(* PLC project PLCopen TC4 OPC UA, University of Seoul OPC UA 0.0 *)
(* stored: creationDateTime 2015-10-01T00:00:00, modificationDateTime 2015-10-01T00:00:00 *)

TYPE UASecurityMsgMode : (UASMM_BestAvailable, UASMM_None, UASMM_Sign, UASMM_SignEncrypt);
END_TYPE

TYPE UASecurityPolicy : (UASP_BestAvailable, UASP_None, UASP_Basic128Rsa15, UASP_Basic256, UASP_Basic256Sha256);
END_TYPE

TYPE UATransportProfile : (UATP_UATcp, UATP_WSHttpBinary, UATP_WSHttpXmlOrBinary, UATP_WSHttpXml);
END_TYPE

TYPE UAUserIdentityTokenType : (UAUITT_Anonymous, UAUITT_Username, UAUITT_x509, UAUITT_IssuedToken);
END_TYPE

TYPE UAIdentifierType : (UAIT_Numeric, UAIT_String, UAIT_GUID, UAIT_Opaque);
END_TYPE

TYPE UADeadbandType : (UADT_None, UADT_Absolute, UADT_Percent) := UADT_None;
END_TYPE

TYPE UAAttributeID : (UAAI_NodeID, UAAI_NodeClass, UAAI_BrowseName, UAAI_DisplayName, UAAI_Description, UAAI_WriteMask, UAAI_UserWriteMask, UAAI_IsAbstract, UAAI_Symmetric, UAAI_InverseName, UAAI_ContainsNoLoops, UAAI_EventNotifier, UAAI_Value, UAAI_DataType, UAAI_ValueRank, UAAI_ArrayDimensions, UAAI_AccessLevel, UAAI_UserAccessLevel, UAAI_MinimumSamplingInterval, UAAI_Historizing, UAAI_Executable, UAAI_UserExecutable) := UAAI_NodeID;
END_TYPE

TYPE UAConnectionStatus : (UACS_Connected, UACS_ConnectionError, UACS_Shutdown);
END_TYPE

TYPE UAServerState : (UASS_Running, UASS_Failed, UASS_NoConfiguration, UASS_Suspended, UASS_Shutdown, UASS_Test, UASS_CommunicationFault, UASS_Unknown);
END_TYPE

TYPE UANodeClassMask : (UANCM_None, UANCM_Object, UANCM_Variable, UANCM_Method, UANCM_ObjectType, UANCM_VariableType, UANCM_ReferenceType, UANCM_DataType, UANCM_View, UANCM_All);
END_TYPE

TYPE _UA_VariantType : (PlcOpen_VariantType_Boolaen, PlcOpen_VariantType_Byte, PlcOpen_VariantType_CharA, PlcOpen_VariantType_Int16, PlcOpen_VariantType_Int32, PlcOpen_VariantType_UInt16, PlcOpen_VariantType_UInt32, PlcOpen_VariantType_Double, PlcOpen_VariantType_Float, PlcOpen_VariantType_StringA, PlcOpen_VariantType_DateTime, PlcOpen_VariantType_QualifiedName);
END_TYPE

TYPE UAUserIdentityToken : STRUCT
  UserIdentityTokenType : UAUserIdentityTokenType;
  TokenParam1 : STRING;
  TokenParam2 : STRING;
END_STRUCT;
END_TYPE

TYPE UASessionConnectInfo : STRUCT
  SessionName : STRING;
  ApplicationName : STRING;
  SecurityMsgMode : UASecurityMsgMode;
  SecurityPolicy : UASecurityPolicy;
  CertificateStore : STRING;
  ClientCertificateName : STRING;
  ServerUri : STRING;
  CheckServerCertificate : BOOL;
  TransportProfile : UATransportProfile;
  UserIdentityToken : UAUserIdentityToken;
  VendorSpecificParameter : STRING;
  SessionTimeout : STRING;
  MonitorConnection : STRING;
  LocaleIDs : STRING;
END_STRUCT;
END_TYPE

TYPE UANODEID : STRUCT
  NamespaceIndex : UINT;
  Identifier : STRING;
  IdentifierType : UAIdentifierType;
END_STRUCT;
END_TYPE

TYPE UAQualifiedName : STRUCT
  NamespaceIndex : UINT;
  Name : STRING;
END_STRUCT;
END_TYPE

TYPE UAMONITORINGPARAMETER : STRUCT
  SamplingInterval : STRING;
  QueueSize : UINT;
  DiscardOldest : BOOL;
  DeadbandType : UADeadbandType;
  Deadband : REAL;
END_STRUCT;
END_TYPE

TYPE UALocalizedText : STRUCT
  Locale : _UALocaleType;
  Text : STRING;
END_STRUCT;
END_TYPE

TYPE UANodeInformation : STRUCT
  AccessLevel : BYTE;
  ArrayDimension : _UA_UDINT_ArrayType;
  BrowseName : UAQualifiedName;
  ContainsNoLoops : BOOL;
  DataType : UANODEID;
  Description : UALocalizedText;
  DisplayName : UALocalizedText;
  EventNotifier : BYTE;
  Executable : BOOL;
  Historizing : BOOL;
  InverseName : STRING;
  IsAbstract : BOOL;
  MinimumSamplingInterval : STRING;
  NodeClass : UANodeClassMask;
  Symmetric : BOOL;
  UserAccessLevel : BYTE;
  UserExecutable : BOOL;
  UserWriteMask : UDINT;
  ValueRank : DINT;
  WriteMask : UDINT;
END_STRUCT;
END_TYPE

TYPE UAINDEXRANGE : STRUCT
  StartIndex : UINT;
  EndIndex : UINT;
END_STRUCT;
END_TYPE

TYPE UANODEADDITIONALINFO : STRUCT
  AttributeID : UAAttributeID;
  IndexRangeCount : UINT;
  IndexRange : ARRAY[1..20] OF UAINDEXRANGE;
END_STRUCT;
END_TYPE

TYPE _UA_BOOL_ArrayType : STRUCT
  Elements : ARRAY[1..20] OF BOOL;
END_STRUCT;
END_TYPE

TYPE _UA_UINT_ArrayType : STRUCT
  Elements : ARRAY[1..20] OF UINT;
END_STRUCT;
END_TYPE

TYPE _UA_UDINT_ArrayType : STRUCT
  Elements : ARRAY[1..20] OF UDINT;
END_STRUCT;
END_TYPE

TYPE _UA_DT_ArrayType : STRUCT
  Elements : ARRAY[1..20] OF STRING;
END_STRUCT;
END_TYPE

TYPE _UA_STRING_ArrayType : STRUCT
  Elements : ARRAY[1..20] OF STRING;
END_STRUCT;
END_TYPE

TYPE _UA_DWORD_ArrayType : STRUCT
  Elements : ARRAY[1..20] OF DWORD;
END_STRUCT;
END_TYPE

TYPE _UA_UANODEID_ArrayType : STRUCT
  Elements : ARRAY[1..20] OF UANODEID;
END_STRUCT;
END_TYPE

TYPE _UA_MONITORINGPARAMETER_ArrayType : STRUCT
  Elements : ARRAY[1..20] OF UAMONITORINGPARAMETER;
END_STRUCT;
END_TYPE

TYPE _UA_NODEADDITIONALINFO_ArrayType : STRUCT
  Elements : ARRAY[1..20] OF UANODEADDITIONALINFO;
END_STRUCT;
END_TYPE

TYPE _UA_METHODARGUMENT_ArrayType : STRUCT
  Elements : ARRAY[1..20] OF _UA_METHODARGUMENT;
END_STRUCT;
END_TYPE

TYPE _UALocaleType : STRUCT
  Locale : ARRAY[1..5] OF STRING;
END_STRUCT;
END_TYPE

TYPE _UA_METHODARGUMENT : STRUCT
  VariantType : _UA_VariantType;
  Value : STRING;
END_STRUCT;
END_TYPE

TYPE _UA_MethodParameter : STRUCT
  NoOfArgument : UINT;
  Arguments : _UA_METHODARGUMENT_ArrayType;
END_STRUCT;
END_TYPE

FUNCTION_BLOCK UA_Connect
  VAR_INPUT
    Execute : BOOL := FALSE;
    ServerEndpointUrl : STRING;
    SessionConnectInfo : UASessionConnectInfo;
    Timeout : TIME;
  END_VAR
  VAR_OUTPUT
    ConnectionHdl : DWORD;
    Done : BOOL := FALSE;
    Busy : BOOL := FALSE;
    Error : BOOL := FALSE;
    ErrorID : DWORD;
  END_VAR
  VAR
    State : DWORD;
    Trigm1 : BOOL := FALSE;
    Trigged : BOOL := FALSE;
    Pre_ServerEndpointUrl : STRING;
    Pre_ServerEndpointUrl0 : STRING;
    Pre_SessionConnectInfo : UASessionConnectInfo;
    Pre_SessionConnectInfo0 : UASessionConnectInfo;
    Pre_Timeout : TIME;
    Pre_Timeout0 : TIME;
    Pre_ConnectionHdl : DWORD;
    Pre_ErrorID : DWORD;
  END_VAR

{{
  #ifdef _ENABLE_OPC_UA_CLIENT
  extern void __UA_ConnectFB(UA_CONNECT*);
  __UA_ConnectFB(data__);
  #endif
}}
          
END_FUNCTION_BLOCK

FUNCTION_BLOCK UA_Disconnect
  VAR_INPUT
    Execute : BOOL;
    ConnectionHdl : DWORD;
    Timeout : TIME;
  END_VAR
  VAR_OUTPUT
    Done : BOOL;
    Busy : BOOL;
    Error : BOOL;
    ErrorID : DWORD;
  END_VAR
  VAR
    State : DWORD;
    Trigm1 : BOOL;
    Trigged : BOOL;
    Pre_ConnectionHdl : DWORD;
    Pre_ConnectionHdl0 : DWORD;
    Pre_Timeout : TIME;
    Pre_Timeout0 : TIME;
    Pre_ErrorID : DWORD;
  END_VAR

{{
  #ifdef _ENABLE_OPC_UA_CLIENT
  extern void __UA_DisconnectFB(UA_DISCONNECT*);
  __UA_DisconnectFB(data__);
  #endif
}}
          
END_FUNCTION_BLOCK

FUNCTION_BLOCK UA_NamespaceGetIndexList
  VAR_INPUT
    Execute : BOOL;
    ConnectionHdl : DWORD;
    NamespaceUrisCount : UINT;
    NamespaceUris : _UA_STRING_ArrayType;
    Timeout : TIME;
  END_VAR
  VAR_OUTPUT
    NamespaceIndexes : _UA_UINT_ArrayType;
    Done : BOOL;
    Busy : BOOL;
    Error : BOOL;
    ErrorID : DWORD;
    ErrorIDs : ARRAY[1..50] OF DWORD;
  END_VAR
  VAR
    State : DWORD;
    Trigm1 : BOOL;
    Trigged : BOOL;
    Pre_ConnectionHdl : DWORD;
    Pre_ConnectionHdl0 : DWORD;
    Pre_NamespaceUrisCount : UINT;
    Pre_NamespaceUrisCount0 : UINT;
    Pre_NamespaceUris : _UA_STRING_ArrayType;
    Pre_NamespaceUris0 : _UA_STRING_ArrayType;
    Pre_NamespaceIndexes : _UA_UINT_ArrayType;
    Pre_Timeout : TIME;
    Pre_Timeout0 : TIME;
    Pre_ErrorID : DWORD;
  END_VAR

{{
  #ifdef _ENABLE_OPC_UA_CLIENT
  extern void __UA_NamespaceGetIndexListFB(UA_NAMESPACEGETINDEXLIST*);
  __UA_NamespaceGetIndexListFB(data__);
  #endif
}}
          
END_FUNCTION_BLOCK

FUNCTION_BLOCK UA_NodeGetHandleList
  VAR_INPUT
    Execute : BOOL;
    ConnectionHdl : DWORD;
    NodeIDCount : UINT;
    NodeIDs : _UA_UANODEID_ArrayType;
    Timeout : TIME;
  END_VAR
  VAR_OUTPUT
    NodeHdls : _UA_DWORD_ArrayType;
    Done : BOOL;
    Busy : BOOL;
    Error : BOOL;
    ErrorID : DWORD;
    NodeErrorIDs : ARRAY[1..20] OF DWORD;
  END_VAR
  VAR
    State : DWORD;
    Trigm1 : BOOL;
    Trigged : BOOL;
    Pre_ConnectionHdl : DWORD;
    Pre_ConnectionHdl0 : DWORD;
    Pre_NodeIDCount : UINT;
    Pre_NodeIDCount0 : UINT;
    Pre_NodeIDs : _UA_UANODEID_ArrayType;
    Pre_NodeIDs0 : _UA_UANODEID_ArrayType;
    Pre_Timeout : TIME;
    Pre_Timeout0 : TIME;
    Pre_NodeHdls : _UA_DWORD_ArrayType;
    Pre_ErrorID : DWORD;
    Pre_NodeErrorIDs : ARRAY[1..20] OF DWORD;
  END_VAR

{{
  #ifdef _ENABLE_OPC_UA_CLIENT
  extern void __UA_NodeGetHandleListFB(UA_NODEGETHANDLELIST*);
  __UA_NodeGetHandleListFB(data__);
  #endif
}}
          
END_FUNCTION_BLOCK

FUNCTION_BLOCK UA_NodeReleaseHandleList
  VAR_INPUT
    Execute : BOOL;
    ConnectionHdl : DWORD;
    NodeHdlCount : UINT;
    NodeHdls : _UA_DWORD_ArrayType;
    Timeout : TIME;
  END_VAR
  VAR_OUTPUT
    Done : BOOL;
    Busy : BOOL;
    Error : BOOL;
    ErrorID : DWORD;
    NodeErrorIDs : ARRAY[1..20] OF DWORD;
  END_VAR
  VAR
    State : DWORD;
    Trigm1 : BOOL;
    Trigged : BOOL;
    Pre_ConnectionHdl : DWORD;
    Pre_ConnectionHdl0 : DWORD;
    Pre_NodeHdlCount : UINT;
    Pre_NodeHdlCount0 : UINT;
    Pre_NodeHdls : _UA_DWORD_ArrayType;
    Pre_NodeHdls0 : _UA_DWORD_ArrayType;
    Pre_Timeout : TIME;
    Pre_Timeout0 : TIME;
    Pre_ErrorID : DWORD;
    Pre_NodeErrorIDs : ARRAY[1..20] OF DWORD;
  END_VAR

{{
  #ifdef _ENABLE_OPC_UA_CLIENT
  extern void __UA_NodeReleaseHandleListFB(UA_NODERELEASEHANDLELIST*);
  __UA_NodeReleaseHandleListFB(data__);
  #endif
}}
          
END_FUNCTION_BLOCK

FUNCTION_BLOCK UA_NodeGetInformation
  VAR_INPUT
    Execute : BOOL;
    ConnectionHdl : DWORD;
    NodeID : UANODEID;
    Timeout : TIME;
  END_VAR
  VAR_OUTPUT
    NodeInfo : UANodeInformation;
    Done : BOOL;
    Busy : BOOL;
    Error : BOOL;
    NodeGetInfoErrorIDs : ARRAY[0..21] OF DWORD;
  END_VAR
  VAR
    State : BOOL;
    Trigm1 : BOOL;
    Trigged : BOOL;
    Pre_ConnectionHdl : DWORD;
    Pre_ConnectionHdl0 : DWORD;
    Pre_NodeID : UANODEID;
    Pre_NodeID0 : UANODEID;
    Pre_Timeout : TIME;
    Pre_Timeout0 : TIME;
    Pre_NodeInfo : UANodeInformation;
    Pre_NodeGetInfoErrorIDs : ARRAY[0..21] OF DWORD;
    ErrorID : DWORD;
  END_VAR

{{
  #ifdef _ENABLE_OPC_UA_CLIENT
  extern void __UA_NodeGetInformationFB(UA_NODEGETINFORMATION*);
  __UA_NodeGetInformationFB(data__);
  #endif
}}
          
END_FUNCTION_BLOCK

FUNCTION_BLOCK UA_SubscriptionCreate
  VAR_INPUT
    Execute : BOOL;
    ConnectionHdl : DWORD;
    PublishingEnable : BOOL;
    Priority : BYTE;
    Timeout : TIME;
  END_VAR
  VAR_OUTPUT
    SubscriptionHdl : DWORD;
    Done : BOOL;
    Busy : BOOL;
    Error : BOOL;
    ErrorID : DWORD;
  END_VAR
  VAR_IN_OUT
    PublishingInterval : TIME;
  END_VAR
  VAR
    State : DWORD;
    Trigm1 : BOOL;
    Trigged : BOOL;
    Pre_ConnectionHdl : DWORD;
    Pre_ConnectionHdl0 : DWORD;
    Pre_PublishingEnable : BOOL;
    Pre_PublishingEnable0 : BOOL;
    Pre_Priority : BYTE;
    Pre_Priority0 : BYTE;
    Pre_Timeout : TIME;
    Pre_Timeout0 : TIME;
    Pre_PublishingInterval : TIME;
    Pre_PublishingInterval0 : TIME;
    Pre_PublishingInterval1 : TIME;
    Pre_SubscriptionHdl : DWORD;
    Pre_SubscriptionHdl0 : DWORD;
    Pre_ErrorID : DWORD;
    Pre_ErrorID0 : DWORD;
  END_VAR

{{
  #ifdef _ENABLE_OPC_UA_CLIENT
  extern void __UA_SubscriptionCreateFB(UA_SUBSCRIPTIONCREATE*);
  __UA_SubscriptionCreateFB(data__);
  #endif
}}
          
END_FUNCTION_BLOCK

FUNCTION_BLOCK UA_SubscriptionDelete
  VAR_INPUT
    Execute : BOOL;
    SubscriptionHdl : DWORD;
    Timeout : TIME;
  END_VAR
  VAR_OUTPUT
    Done : BOOL;
    Busy : BOOL;
    Error : BOOL;
    ErrorID : DWORD;
  END_VAR
  VAR
    State : DWORD;
    Trigm1 : BOOL;
    Trigged : BOOL;
    Pre_SubscriptionHdl : DWORD;
    Pre_SubscriptionHdl0 : DWORD;
    Pre_Timeout : TIME;
    Pre_Timeout0 : TIME;
    Pre_ErrorID : DWORD;
  END_VAR

{{
  #ifdef _ENABLE_OPC_UA_CLIENT
  extern void __UA_SubscriptionDeleteFB(UA_SUBSCRIPTIONDELETE*);
  __UA_SubscriptionDeleteFB(data__);
  #endif

}}
          
END_FUNCTION_BLOCK

FUNCTION_BLOCK UA_SubscriptionProcessed
  VAR_INPUT
    Execute : BOOL;
    SubscriptionHdl : DWORD;
  END_VAR
  VAR
    Pre_SubscriptionHdl : DWORD;
    Pre_SubscriptionHdl0 : DWORD;
  END_VAR
  VAR_INPUT
    Timeout : TIME;
  END_VAR
  VAR
    Pre_Timeout : TIME;
    Pre_Timeout0 : TIME;
  END_VAR
  VAR_OUTPUT
    Published : BOOL;
  END_VAR
  VAR
    Pre_Published : BOOL;
  END_VAR
  VAR_OUTPUT
    Done : BOOL;
    Busy : BOOL;
    Error : BOOL;
    ErrorID : DWORD;
  END_VAR
  VAR
    Pre_ErrorID : DWORD;
    State : DWORD;
    Trigged : BOOL;
    Trigm1 : BOOL;
  END_VAR

{{
  #ifdef _ENABLE_OPC_UA_CLIENT
  extern void __UA_SubscriptionProcessedFB(UA_SUBSCRIPTIONPROCESSED*);
  __UA_SubscriptionProcessedFB(data__);
  #endif
}}
          
END_FUNCTION_BLOCK

FUNCTION_BLOCK UA_MonitoredItemAddList
  VAR_INPUT
    Execute : BOOL;
    SubscriptionHdl : DWORD;
  END_VAR
  VAR
    Pre_SubscriptionHdl : DWORD;
    Pre_SubscriptionHdl0 : DWORD;
  END_VAR
  VAR_INPUT
    NodeHdlCount : UINT;
  END_VAR
  VAR
    Pre_NodeHdlCount : UINT;
    Pre_NodeHdlCount0 : UINT;
  END_VAR
  VAR_INPUT
    NodeHdls : _UA_DWORD_ArrayType;
  END_VAR
  VAR
    Pre_NodeHdls : _UA_DWORD_ArrayType;
    Pre_NodeHdls0 : _UA_DWORD_ArrayType;
  END_VAR
  VAR_INPUT
    NodeAddInfos : _UA_NodeAdditionalInfo_ArrayType;
  END_VAR
  VAR
    Pre_NodeAddInfos : _UA_NodeAdditionalInfo_ArrayType;
    Pre_NodeAddInfos0 : _UA_NodeAdditionalInfo_ArrayType;
  END_VAR
  VAR_INPUT
    Timeout : TIME;
  END_VAR
  VAR
    Pre_Timeout : TIME;
    Pre_Timeout0 : TIME;
  END_VAR
  VAR_OUTPUT
    Done : BOOL;
    Busy : BOOL;
    Error : BOOL;
    ErrorID : DWORD;
  END_VAR
  VAR
    Pre_ErrorID : DWORD;
  END_VAR
  VAR_OUTPUT
    NodeErrorIDs : _UA_DWORD_ArrayType;
  END_VAR
  VAR
    Pre_NodeErrorIDs : _UA_DWORD_ArrayType;
  END_VAR
  VAR_OUTPUT
    MonitoredItemHdls : _UA_DWORD_ArrayType;
  END_VAR
  VAR
    Pre_MonitoredItemHdls : _UA_DWORD_ArrayType;
  END_VAR
  VAR_IN_OUT
    Variables : UINT;
  END_VAR
  VAR
    Pre_Variables : UINT;
    Pre_Variables0 : UINT;
    Pre_Variables1 : UINT;
  END_VAR
  VAR_IN_OUT
    MonitoringSettings : _UA_MONITORINGPARAMETER_ArrayType;
  END_VAR
  VAR
    Pre_MonitoringSettings : _UA_MONITORINGPARAMETER_ArrayType;
    Pre_MonitoringSettings0 : _UA_MONITORINGPARAMETER_ArrayType;
    Pre_MonitoringSettings1 : _UA_MONITORINGPARAMETER_ArrayType;
  END_VAR
  VAR_IN_OUT
    ValuesChanged : UINT;
  END_VAR
  VAR
    Pre_ValuesChanged : UINT;
    Pre_ValuesChanged0 : UINT;
    Pre_ValuesChanged1 : UINT;
  END_VAR
  VAR_IN_OUT
    RemainingValueCount : _UA_UINT_ArrayType;
  END_VAR
  VAR
    Pre_RemainingValueCount : _UA_UINT_ArrayType;
    Pre_RemainingValueCount0 : _UA_UINT_ArrayType;
    Pre_RemainingValueCount1 : _UA_UINT_ArrayType;
  END_VAR
  VAR_IN_OUT
    TimeStamps : _UA_DT_ArrayType;
  END_VAR
  VAR
    Pre_TimeStamps : _UA_DT_ArrayType;
    Pre_TimeStamps0 : _UA_DT_ArrayType;
    Pre_TimeStamps1 : _UA_DT_ArrayType;
  END_VAR
  VAR_IN_OUT
    NodeQualityIDs : _UA_DWORD_ArrayType;
  END_VAR
  VAR
    Pre_NodeQualityIDs : _UA_DWORD_ArrayType;
    Pre_NodeQualityIDs0 : _UA_DWORD_ArrayType;
    Pre_NodeQualityIDs1 : _UA_DWORD_ArrayType;
    State : DWORD;
    Trigm1 : BOOL;
    Trigged : BOOL;
  END_VAR

{{
  #ifdef _ENABLE_OPC_UA_CLIENT
  extern void __UA_MonitoredItemAddListFB(UA_MONITOREDITEMADDLIST*);
  __UA_MonitoredItemAddListFB(data__);
  #endif
}}
          
END_FUNCTION_BLOCK

FUNCTION_BLOCK UA_MonitoredItemRemoveList
  VAR_INPUT
    Execute : BOOL;
    SubscriptionHdl : DWORD;
  END_VAR
  VAR
    Pre_SubscriptionHdl : DWORD;
    Pre_SubscriptionHdl0 : DWORD;
  END_VAR
  VAR_INPUT
    MonitoredItemHdlCount : UINT;
  END_VAR
  VAR
    Pre_MonitoredItemHdlCount : UINT;
    Pre_MonitoredItemHdlCount0 : UINT;
  END_VAR
  VAR_INPUT
    MonitoredItemHdls : _UA_DWORD_ArrayType;
  END_VAR
  VAR
    Pre_MonitoredItemHdls : _UA_DWORD_ArrayType;
    Pre_MonitoredItemHdls0 : _UA_DWORD_ArrayType;
  END_VAR
  VAR_INPUT
    Timeout : TIME;
  END_VAR
  VAR
    Pre_Timeout : TIME;
    Pre_Timeout0 : TIME;
  END_VAR
  VAR_OUTPUT
    Done : BOOL;
    Busy : BOOL;
    Error : BOOL;
    ErrorID : DWORD;
  END_VAR
  VAR
    Pre_ErrorID : DWORD;
  END_VAR
  VAR_OUTPUT
    NodeErrorIDs : _UA_DWORD_ArrayType;
  END_VAR
  VAR
    Pre_NodeErrorIDs : _UA_DWORD_ArrayType;
    State : DWORD;
    Trigm1 : BOOL;
    Trigged : BOOL;
  END_VAR

{{
  #ifdef _ENABLE_OPC_UA_CLIENT
  extern void __UA_MonitoredItemRemoveListFB(UA_MONITOREDITEMREMOVELIST*);
  __UA_MonitoredItemRemoveListFB(data__);
  #endif
}}
          
END_FUNCTION_BLOCK

FUNCTION_BLOCK UA_MonitoredItemOperateList
  VAR_INPUT
    Enable : BOOL;
    SubscriptionHdl : DWORD;
  END_VAR
  VAR
    Pre_SubscriptionHdl : DWORD;
    Pre_SubscriptionHdl0 : DWORD;
  END_VAR
  VAR_INPUT
    MonitoredItemHdlCount : UINT;
  END_VAR
  VAR
    Pre_MonitoredItemHdlCount : UINT;
    Pre_MonitoredItemHdlCount0 : UINT;
  END_VAR
  VAR_INPUT
    MonitoredItemHdls : _UA_DWORD_ArrayType;
  END_VAR
  VAR
    Pre_MonitoredItemHdls : _UA_DWORD_ArrayType;
    Pre_MonitoredItemHdls0 : _UA_DWORD_ArrayType;
  END_VAR
  VAR_OUTPUT
    Published : BOOL;
  END_VAR
  VAR
    Pre_Published : BOOL;
  END_VAR
  VAR_OUTPUT
    Done : BOOL;
    Busy : BOOL;
    Error : BOOL;
    ErrorID : DWORD;
  END_VAR
  VAR
    Pre_ErrorID : DWORD;
    State : DWORD;
    Trigm1 : BOOL;
    Trigged : BOOL;
  END_VAR

{{
  #ifdef _ENABLE_OPC_UA_CLIENT
  extern void __UA_MonitoredItemOperateListFB(UA_MONITOREDITEMOPERATELIST*);
  __UA_MonitoredItemOperateListFB(data__);
  #endif
}}
          
END_FUNCTION_BLOCK

FUNCTION_BLOCK UA_ReadList
  VAR_INPUT
    Execute : BOOL;
    ConnectionHdl : DWORD;
    NodeHdlCount : UINT;
    NodeHdls : _UA_DWORD_ArrayType;
    NodeAddInfos : ARRAY[1..20] OF UANODEADDITIONALINFO;
    Timeout : TIME;
  END_VAR
  VAR_OUTPUT
    Done : BOOL;
    Busy : BOOL;
    Error : BOOL;
    ErrorID : DWORD;
    NodeErrorIDs : ARRAY[1..20] OF DWORD;
    TimeStamps : ARRAY[1..20] OF STRING;
  END_VAR
  VAR_IN_OUT
    Variables : _UA_STRING_ArrayType;
  END_VAR
  VAR
    State : DWORD;
    Trigm1 : BOOL;
    Trigged : BOOL;
    Pre_ConnectionHdl : DWORD;
    Pre_ConnectionHdl0 : DWORD;
    Pre_NodeHdlCount : UINT;
    Pre_NodeHdlCount0 : UINT;
    Pre_NodeHdls : _UA_DWORD_ArrayType;
    Pre_NodeHdls0 : _UA_DWORD_ArrayType;
    Pre_NodeAddInfos : ARRAY[1..20] OF UANODEADDITIONALINFO;
    Pre_NodeAddInfos0 : ARRAY[1..20] OF UANODEADDITIONALINFO;
    Pre_Timeout : TIME;
    Pre_Timeout0 : TIME;
    Pre_ErrorID : DWORD;
    Pre_NodeErrorIDs : ARRAY[1..20] OF DWORD;
    Pre_TimeStamps : ARRAY[1..20] OF STRING;
    Pre_Variables : _UA_STRING_ArrayType;
  END_VAR

{{
  #ifdef _ENABLE_OPC_UA_CLIENT
  extern void __UA_ReadListFB(UA_READLIST*);
  __UA_ReadListFB(data__);
  #endif
}}
          
END_FUNCTION_BLOCK

FUNCTION_BLOCK UA_WriteList
  VAR_INPUT
    Execute : BOOL;
    ConnectionHdl : DWORD;
    NodeHdlCount : UINT;
    NodeHdls : _UA_DWORD_ArrayType;
    NodeAddInfos : ARRAY[1..20] OF UANODEADDITIONALINFO;
    Timeout : TIME;
  END_VAR
  VAR_OUTPUT
    Done : BOOL;
    Busy : BOOL;
    Error : BOOL;
    ErrorID : DWORD;
    NodeErrorIDs : ARRAY[1..20] OF DWORD;
  END_VAR
  VAR_IN_OUT
    Variables : _UA_STRING_ArrayType;
  END_VAR
  VAR
    State : DWORD;
    Trigm1 : BOOL;
    Trigged : BOOL;
    Pre_ConnectionHdl : DWORD;
    Pre_ConnectionHdl0 : DWORD;
    Pre_NodeHdlCount : UINT;
    Pre_NodeHdlCount0 : UINT;
    Pre_NodeHdls : _UA_DWORD_ArrayType;
    Pre_NodeHdls0 : _UA_DWORD_ArrayType;
    Pre_NodeAddInfos : ARRAY[1..20] OF UANODEADDITIONALINFO;
    Pre_NodeAddInfos0 : ARRAY[1..20] OF UANODEADDITIONALINFO;
    Pre_Timeout : TIME;
    Pre_Timeout0 : TIME;
    Pre_Variables : _UA_STRING_ArrayType;
    Pre_Variables0 : _UA_STRING_ArrayType;
    Pre_ErrorID : DWORD;
    Pre_NodeErrorIDs : ARRAY[1..20] OF DWORD;
  END_VAR

{{
  #ifdef _ENABLE_OPC_UA_CLIENT
  extern void __UA_WriteListFB(UA_WRITELIST*);
  __UA_WriteListFB(data__);
  #endif
}}
          
END_FUNCTION_BLOCK

FUNCTION_BLOCK UA_MethodGetHandleList
  VAR_INPUT
    Execute : BOOL;
    ConnectionHdl : DWORD;
  END_VAR
  VAR
    Pre_ConnectionHdl : DWORD;
    Pre_ConnectionHdl0 : DWORD;
  END_VAR
  VAR_INPUT
    NodeIDCount : UINT;
  END_VAR
  VAR
    Pre_NodeIDCount : UINT;
    Pre_NodeIDCount0 : UINT;
  END_VAR
  VAR_INPUT
    ObjectNodeIDs : _UA_UANODEID_ArrayType;
  END_VAR
  VAR
    Pre_ObjectNodeIDs : _UA_UANODEID_ArrayType;
    Pre_ObjectNodeIDs0 : _UA_UANODEID_ArrayType;
  END_VAR
  VAR_INPUT
    MethodNodeIDs : _UA_UANODEID_ArrayType;
  END_VAR
  VAR
    Pre_MethodNodeIDs : _UA_UANODEID_ArrayType;
    Pre_MethodNodeIDs0 : _UA_UANODEID_ArrayType;
  END_VAR
  VAR_INPUT
    Timeout : TIME;
  END_VAR
  VAR
    Pre_Timeout : TIME;
    Pre_Timeout0 : TIME;
  END_VAR
  VAR_OUTPUT
    MethodHdls : _UA_DWORD_ArrayType;
  END_VAR
  VAR
    Pre_MethodHdls : _UA_DWORD_ArrayType;
  END_VAR
  VAR_OUTPUT
    Done : BOOL;
    Busy : BOOL;
    Error : BOOL;
    ErrorIDs : _UA_DWORD_ArrayType;
  END_VAR
  VAR
    Pre_ErrorIDs : _UA_DWORD_ArrayType;
    State : DWORD;
    Trigged : BOOL;
    Trigm1 : BOOL;
  END_VAR

{{
  #ifdef _ENABLE_OPC_UA_CLIENT
  extern void __UA_MethodGetHandleListFB(UA_METHODGETHANDLELIST*);
  __UA_MethodGetHandleListFB(data__);
  #endif
}}
          
END_FUNCTION_BLOCK

FUNCTION_BLOCK UA_MethodReleaseHandleList
  VAR_INPUT
    Execute : BOOL;
    ConnectionHdl : DWORD;
  END_VAR
  VAR
    Pre_ConnectionHdl : DWORD;
    Pre_ConnectionHdl0 : DWORD;
  END_VAR
  VAR_INPUT
    MethodHdlCount : UINT;
  END_VAR
  VAR
    Pre_MethodHdlCount : UINT;
    Pre_MethodHdlCount0 : UINT;
  END_VAR
  VAR_INPUT
    MethodHdls : _UA_DWORD_ArrayType;
  END_VAR
  VAR
    Pre_MethodHdls : _UA_DWORD_ArrayType;
    Pre_MethodHdls0 : _UA_DWORD_ArrayType;
  END_VAR
  VAR_INPUT
    Timeout : TIME;
  END_VAR
  VAR
    Pre_Timeout : TIME;
    Pre_Timeout0 : TIME;
  END_VAR
  VAR_OUTPUT
    Done : BOOL;
    Busy : BOOL;
    Error : BOOL;
    ErrorIDs : _UA_DWORD_ArrayType;
  END_VAR
  VAR
    Pre_ErrorIDs : _UA_DWORD_ArrayType;
    Pre_ErrorIDs0 : _UA_DWORD_ArrayType;
    State : DWORD;
    Trigm1 : BOOL;
    Trigged : BOOL;
  END_VAR

{{
  #ifdef _ENABLE_OPC_UA_CLIENT
  extern void __UA_MethodReleaseHandleListFB(UA_METHODRELEASEHANDLELIST*);
  __UA_MethodReleaseHandleListFB(data__);
  #endif
}}
          
END_FUNCTION_BLOCK

FUNCTION_BLOCK UA_MethodCall
  VAR_INPUT
    Execute : BOOL;
    ConnectionHdl : DWORD;
  END_VAR
  VAR
    Pre_ConnectionHdl : DWORD;
    Pre_ConnectionHdl0 : DWORD;
  END_VAR
  VAR_INPUT
    MethodHdl : DWORD;
  END_VAR
  VAR
    Pre_MethodHdl : DWORD;
    Pre_MethodHdl0 : DWORD;
  END_VAR
  VAR_INPUT
    Timeout : TIME;
  END_VAR
  VAR
    Pre_Timeout : TIME;
    Pre_Timeout0 : TIME;
  END_VAR
  VAR_OUTPUT
    Done : BOOL;
    Busy : BOOL;
    Error : BOOL;
    ErrorID : DWORD;
  END_VAR
  VAR
    Pre_ErrorID : DWORD;
  END_VAR
  VAR_IN_OUT
    InputArguments : _UA_MethodParameter;
  END_VAR
  VAR
    Pre_InputArguments : _UA_MethodParameter;
    Pre_InputArguments0 : _UA_MethodParameter;
    Pre_InputArguments1 : _UA_MethodParameter;
  END_VAR
  VAR_IN_OUT
    OutputArguments : _UA_MethodParameter;
  END_VAR
  VAR
    Pre_OutputArguments : _UA_MethodParameter;
    Pre_OutputArguments0 : _UA_MethodParameter;
    Pre_OutputArguments1 : _UA_MethodParameter;
    State : DWORD;
    Trigm1 : BOOL;
    Trigged : BOOL;
  END_VAR

{{
  #ifdef _ENABLE_OPC_UA_CLIENT
  extern void __UA_MethodCallFB(UA_METHODCALL*);
  __UA_MethodCallFB(data__);
  #endif
}}
          
END_FUNCTION_BLOCK

FUNCTION_BLOCK UA_ConnectionGetStatus
  VAR_INPUT
    Execute : BOOL;
    ConnectionHdl : DWORD;
  END_VAR
  VAR
    Pre_ConnectionHdl : DWORD;
    Pre_ConnectionHdl0 : DWORD;
  END_VAR
  VAR_INPUT
    Timeout : TIME;
  END_VAR
  VAR
    Pre_Timeout : TIME;
    Pre_Timeout0 : TIME;
  END_VAR
  VAR_OUTPUT
    ConnectionStatus : UAConnectionStatus;
  END_VAR
  VAR
    Pre_ConnectionStatus : UAConnectionStatus;
    Pre_ConnectionStatus0 : UAConnectionStatus;
  END_VAR
  VAR_OUTPUT
    ServerState : UAServerState;
  END_VAR
  VAR
    Pre_ServerState : UAServerState;
  END_VAR
  VAR_OUTPUT
    ServiceLevel : BYTE;
  END_VAR
  VAR
    Pre_ServiceLevel : BYTE;
  END_VAR
  VAR_OUTPUT
    Done : BOOL;
    Busy : BOOL;
    Error : BOOL;
    ErrorID : DWORD;
  END_VAR
  VAR
    Pre_ErrorID : DWORD;
    State : DWORD;
    Trigm1 : BOOL;
    Trigged : BOOL;
  END_VAR

{{
  #ifdef _ENABLE_OPC_UA_CLIENT
  extern void __UA_ConnectionGetStatusFB(UA_CONNECTIONGETSTATUS*);
  __UA_ConnectionGetStatusFB(data__);
  #endif
}}
          
END_FUNCTION_BLOCK

FUNCTION_BLOCK _UA_GetDWORDFromArray
  VAR_INPUT
    Enable : BOOL;
  END_VAR
  VAR_OUTPUT
    Done : BOOL;
  END_VAR
  VAR_INPUT
    DWORDarray : _UA_DWORD_ArrayType;
    index : UINT;
  END_VAR
  VAR_OUTPUT
    DWORDvalue : DWORD;
  END_VAR

IF Enable=TRUE THEN
	DWORDvalue:=DWORDarray.Elements[index];
	Done:=TRUE;
END_IF;
IF Enable=FALSE THEN
  Done:=FALSE;
END_IF;
          
END_FUNCTION_BLOCK

FUNCTION_BLOCK _UA_GetUINTFromArray
  VAR_INPUT
    Enable : BOOL;
  END_VAR
  VAR_OUTPUT
    Done : BOOL;
  END_VAR
  VAR_INPUT
    UINTarray : _UA_UINT_ArrayType;
    index : UINT;
  END_VAR
  VAR_OUTPUT
    UINTvalue : UINT;
  END_VAR

IF Enable=TRUE THEN
	UINTvalue:=UINTarray.Elements[index];
	Done:=TRUE;
END_IF;
IF Enable=FALSE THEN
  Done:=FALSE;
END_IF;
          
END_FUNCTION_BLOCK

FUNCTION_BLOCK _UA_GetConnectionStatus
  VAR_INPUT
    Enable : BOOL;
    ConnectionStatus : UAConnectionStatus;
  END_VAR
  VAR_OUTPUT
    Done : BOOL;
    result : STRING;
  END_VAR

IF Enable=TRUE THEN
	CASE ConnectionStatus OF
		UACS_Connected: result:='UACS_Connected';
		UACS_ConnectionError: result:='UACS_ConnectionError';
		UACS_Shutdown: result:='UACS_Shutdown';
	ELSE 
		result:='UACS_ConnectionError';
	END_CASE;
	Done:=TRUE;
END_IF;
IF Enable=FALSE THEN
  Done:=FALSE;
END_IF;
          
END_FUNCTION_BLOCK

FUNCTION_BLOCK _UA_GetServerState
  VAR_INPUT
    Enable : BOOL;
    ServerState : UAServerState;
  END_VAR
  VAR_OUTPUT
    Done : BOOL;
    result : STRING;
  END_VAR

IF Enable=TRUE THEN
	CASE ServerState OF
		UASS_Running: result:='UASS_Running';
		UASS_Failed: result:='UASS_Failed';
		UASS_NoConfiguration: result:='UASS_NoConfiguration';
		UASS_Suspended: result:='UASS_Suspended';
		UASS_Shutdown: result:='UASS_Shutdown';
		UASS_Test: result:='UASS_Test';
		UASS_CommunicationFault: result:='UASS_CommunicationFault';
		UASS_Unknown: result:='UASS_Unknown';
	ELSE 
		result:='UASS_Unknown';
	END_CASE;
	Done:=TRUE;
END_IF;
IF Enable=FALSE THEN
  Done:=FALSE;
END_IF;
          
END_FUNCTION_BLOCK

FUNCTION_BLOCK _UA_GetSessionConnectInfo
  VAR_INPUT
    Enable : BOOL := FALSE;
  END_VAR
  VAR_OUTPUT
    Done : BOOL := FALSE;
  END_VAR
  VAR_INPUT
    SessionName : STRING;
    ApplicationName : STRING;
    SecurityMsgMode : UASecurityMsgMode;
    SecurityPolicy : UASecurityPolicy;
    CertificateStore : STRING;
    ClientCertificateName : STRING;
    ServerUri : STRING;
    CheckServerCertificate : BOOL;
    TransportProfile : UATransportProfile;
    UserIdentityToken : UAUserIdentityToken;
    VendorSpecificParameter : STRING;
    SessionTimeout : STRING;
    MonitorConnection : STRING;
    LocaleIDs : STRING;
  END_VAR
  VAR_OUTPUT
    SessionConnectInfo : UASessionConnectInfo;
  END_VAR

IF Enable=TRUE THEN
	SessionConnectInfo.SessionName:=SessionName;
	SessionConnectInfo.ApplicationName:=ApplicationName;
	SessionConnectInfo.SecurityMsgMode:=SecurityMsgMode;
	SessionConnectInfo.SecurityPolicy:=SecurityPolicy;
	SessionConnectInfo.CertificateStore:=CertificateStore;
	SessionConnectInfo.ClientCertificateName:=ClientCertificateName;
	SessionConnectInfo.ServerUri:=ServerUri;
	SessionConnectInfo.CheckServerCertificate:=CheckServerCertificate;
	SessionConnectInfo.TransportProfile:=TransportProfile;
	SessionConnectInfo.UserIdentityToken:=UserIdentityToken;
	SessionConnectInfo.VendorSpecificParameter:=VendorSpecificParameter;
	SessionConnectInfo.SessionTimeout:=SessionTimeout;
	SessionConnectInfo.MonitorConnection:=MonitorConnection;
	SessionConnectInfo.LocaleIDs:=LocaleIDs;
	Done:=TRUE;
END_IF;
IF Enable=FALSE THEN
  Done:=FALSE;
END_IF;

          
END_FUNCTION_BLOCK

FUNCTION_BLOCK _UA_GetUserIdentityToken
  VAR_INPUT
    Enable : BOOL;
  END_VAR
  VAR_OUTPUT
    Done : BOOL;
  END_VAR
  VAR_INPUT
    UserIdentityTokenType : UAUserIdentityTokenType;
    TokenParam1 : STRING;
    TokenParam2 : STRING;
  END_VAR
  VAR_OUTPUT
    UserIdentityToken : UAUserIdentityToken;
  END_VAR

IF Enable=TRUE THEN
	UserIdentityToken.UserIdentityTokenType:=UserIdentityTokenType;
	UserIdentityToken.TokenParam1:=TokenParam1;
	UserIdentityToken.TokenParam2:=TokenParam2;
	Done:=TRUE;
END_IF;
IF Enable=FALSE THEN
	Done:=FALSE;
END_IF;

          
END_FUNCTION_BLOCK

FUNCTION_BLOCK _UA_GetNamespaceUriArray
  VAR_INPUT
    Enable : BOOL;
  END_VAR
  VAR_OUTPUT
    Done : BOOL;
  END_VAR
  VAR_OUTPUT
    NamespaceUris : _UA_STRING_ArrayType;
  END_VAR
  VAR_INPUT
    NamespaceUri1 : STRING;
    NamespaceUri2 : STRING;
    NamespaceUri3 : STRING;
    NamespaceUri4 : STRING;
    NamespaceUri5 : STRING;
    NamespaceUri6 : STRING;
    NamespaceUri7 : STRING;
    NamespaceUri8 : STRING;
    NamespaceUri9 : STRING;
    NamespaceUri10 : STRING;
    NamespaceUri11 : STRING;
    NamespaceUri12 : STRING;
    NamespaceUri13 : STRING;
    NamespaceUri14 : STRING;
    NamespaceUri15 : STRING;
    NamespaceUri16 : STRING;
    NamespaceUri17 : STRING;
    NamespaceUri18 : STRING;
    NamespaceUri19 : STRING;
    NamespaceUri20 : STRING;
  END_VAR

IF Enable=TRUE THEN
	NamespaceUris.Elements[1] := NamespaceUri1;
	NamespaceUris.Elements[2] := NamespaceUri2;
	NamespaceUris.Elements[3] := NamespaceUri3;
	NamespaceUris.Elements[4] := NamespaceUri4;
	NamespaceUris.Elements[5] := NamespaceUri5;
	NamespaceUris.Elements[6] := NamespaceUri6;
	NamespaceUris.Elements[7] := NamespaceUri7;
	NamespaceUris.Elements[8] := NamespaceUri8;
	NamespaceUris.Elements[9] := NamespaceUri9;
	NamespaceUris.Elements[10] := NamespaceUri10;
	NamespaceUris.Elements[11] := NamespaceUri11;
	NamespaceUris.Elements[12] := NamespaceUri12;
	NamespaceUris.Elements[13] := NamespaceUri13;
	NamespaceUris.Elements[14] := NamespaceUri14;
	NamespaceUris.Elements[15] := NamespaceUri15;
	NamespaceUris.Elements[16] := NamespaceUri16;
	NamespaceUris.Elements[17] := NamespaceUri17;
	NamespaceUris.Elements[18] := NamespaceUri18;
	NamespaceUris.Elements[19] := NamespaceUri19;
	NamespaceUris.Elements[20] := NamespaceUri20;
	Done:=TRUE;
END_IF;
IF Enable=FALSE THEN
  Done:=FALSE;
END_IF;
          
END_FUNCTION_BLOCK

FUNCTION_BLOCK _UA_GetNamespaceIndexResult
  VAR_INPUT
    Enable : BOOL;
  END_VAR
  VAR_OUTPUT
    Done : BOOL;
  END_VAR
  VAR_INPUT
    NamespaceIndexes : _UA_UINT_ArrayType;
    Index : UINT;
  END_VAR
  VAR_OUTPUT
    NamespaceIndex : UINT;
  END_VAR

IF Enable=TRUE THEN
	Done:=FALSE;
	NamespaceIndex := NamespaceIndexes.Elements[index];
	Done:=TRUE;
END_IF;
IF Enable=FALSE THEN
  Done:=FALSE;
END_IF;
          
END_FUNCTION_BLOCK

FUNCTION_BLOCK _UA_GetNodeID
  VAR_INPUT
    Enable : BOOL;
    NamespaceIndex : UINT;
    Identifier : STRING;
    IdentifierType : UAIdentifierType;
  END_VAR
  VAR_OUTPUT
    Done : BOOL;
    NodeID : UANODEID;
  END_VAR
  VAR
    Trigm1 : BOOL;
    Trigged : BOOL;
  END_VAR

IF Enable=TRUE THEN
	NodeID.NamespaceIndex := NamespaceIndex;
	NodeID.Identifier := Identifier;
	NodeID.IdentifierType := IdentifierType;
	Done:=TRUE;
END_IF;
IF Enable=FALSE THEN
  Done:=FALSE;
END_IF;
          
END_FUNCTION_BLOCK

FUNCTION_BLOCK _UA_GetNodeIDArrayFromOne
  VAR_INPUT
    Enable : BOOL;
  END_VAR
  VAR_OUTPUT
    Done : BOOL;
  END_VAR
  VAR_OUTPUT
    NodeIDs : _UA_UANODEID_ArrayType;
  END_VAR
  VAR_INPUT
    NodeID1 : UANODEID;
  END_VAR

IF Enable=TRUE THEN
	NodeIDs.Elements[1] := NodeID1;
	Done:=TRUE;
END_IF;
IF Enable=FALSE THEN
	Done:=FALSE;
END_IF;
          
END_FUNCTION_BLOCK

FUNCTION_BLOCK _UA_GetNodeIDArray
  VAR_INPUT
    Enable : BOOL;
  END_VAR
  VAR_OUTPUT
    Done : BOOL;
  END_VAR
  VAR_OUTPUT
    NodeIDs : _UA_UANODEID_ArrayType;
  END_VAR
  VAR_INPUT
    NodeID1 : UANODEID;
    NodeID2 : UANODEID;
    NodeID3 : UANODEID;
    NodeID4 : UANODEID;
    NodeID5 : UANODEID;
    NodeID6 : UANODEID;
    NodeID7 : UANODEID;
    NodeID8 : UANODEID;
    NodeID9 : UANODEID;
    NodeID10 : UANODEID;
    NodeID11 : UANODEID;
    NodeID12 : UANODEID;
    NodeID13 : UANODEID;
    NodeID14 : UANODEID;
    NodeID15 : UANODEID;
    NodeID16 : UANODEID;
    NodeID17 : UANODEID;
    NodeID18 : UANODEID;
    NodeID19 : UANODEID;
    NodeID20 : UANODEID;
  END_VAR

IF Enable=TRUE THEN
	NodeIDs.Elements[1] := NodeID1;
	NodeIDs.Elements[2] := NodeID2;
	NodeIDs.Elements[3] := NodeID3;
	NodeIDs.Elements[4] := NodeID4;
	NodeIDs.Elements[5] := NodeID5;
	NodeIDs.Elements[6] := NodeID6;
	NodeIDs.Elements[7] := NodeID7;
	NodeIDs.Elements[8] := NodeID8;
	NodeIDs.Elements[9] := NodeID9;
	NodeIDs.Elements[10] := NodeID10;
	NodeIDs.Elements[11] := NodeID11;
	NodeIDs.Elements[12] := NodeID12;
	NodeIDs.Elements[13] := NodeID13;
	NodeIDs.Elements[14] := NodeID14;
	NodeIDs.Elements[15] := NodeID15;
	NodeIDs.Elements[16] := NodeID16;
	NodeIDs.Elements[17] := NodeID17;
	NodeIDs.Elements[18] := NodeID18;
	NodeIDs.Elements[19] := NodeID19;
	NodeIDs.Elements[20] := NodeID20;
	Done:=TRUE;
END_IF;
IF Enable=FALSE THEN
	Done:=FALSE;
END_IF;
          
END_FUNCTION_BLOCK

FUNCTION_BLOCK _UA_GetNodeAdditionalInfo
  VAR_INPUT
    Enable : BOOL;
    NodeInfo : UANodeInformation;
  END_VAR
  VAR_OUTPUT
    Done : BOOL;
    AccessLevel : BYTE;
    ArrayDimension : _UA_UDINT_ArrayType;
    BrowseName : UAQualifiedName;
    ContainsNoLoops : BOOL;
    DataType : UANODEID;
    Description : UALocalizedText;
    DisplayName : UALocalizedText;
    EventNotifier : BYTE;
    Executable : BOOL;
    Historizing : BOOL;
    InverseName : STRING;
    IsAbstract : BOOL;
    MinimumSamplingInterval : STRING;
    NodeClass : UANodeClassMask;
    Symmetric : BOOL;
    UserAccessLevel : BYTE;
    UserExecutable : BOOL;
    UserWriteMask : UDINT;
    ValueRank : DINT;
    WriteMask : UDINT;
  END_VAR

IF Enable=TRUE THEN
	AccessLevel:=NodeInfo.AccessLevel;
	ArrayDimension:=NodeInfo.ArrayDimension;
	BrowseName:=NodeInfo.BrowseName;
	ContainsNoLoops:=NodeInfo.ContainsNoLoops;
	DataType:=NodeInfo.DataType;
	Description:=NodeInfo.Description;
	DisplayName:=NodeInfo.DisplayName;
	EventNotifier:=NodeInfo.EventNotifier;
	Executable:=NodeInfo.Executable;
	Historizing:=NodeInfo.Historizing;
	InverseName:=NodeInfo.InverseName;
	IsAbstract:=NodeInfo.IsAbstract;
	MinimumSamplingInterval:=NodeInfo.MinimumSamplingInterval;
	NodeClass:=NodeInfo.NodeClass;
	Symmetric:=NodeInfo.Symmetric;
	UserAccessLevel:=NodeInfo.UserAccessLevel;
	UserExecutable:=NodeInfo.UserExecutable;
	UserWriteMask:=NodeInfo.UserWriteMask;
	ValueRank:=NodeInfo.ValueRank;
	WriteMask:=NodeInfo.WriteMask;
	Done:=TRUE;
END_IF;
IF Enable=FALSE THEN
	Done:=FALSE;
END_IF;
          
END_FUNCTION_BLOCK

FUNCTION_BLOCK _UA_GetQualifiedName
  VAR_INPUT
    Enable : BOOL;
  END_VAR
  VAR_OUTPUT
    Done : BOOL;
  END_VAR
  VAR_INPUT
    QualifiedName : UAQualifiedName;
  END_VAR
  VAR_OUTPUT
    NamespaceIndex : UINT;
    Name : STRING;
  END_VAR

IF Enable=TRUE THEN
	NamespaceIndex:=QualifiedName.NamespaceIndex;
	Name:=QualifiedName.Name;
	Done:=TRUE;
END_IF;
IF Enable=FALSE THEN
	Done:=FALSE;
END_IF;
          
END_FUNCTION_BLOCK

FUNCTION_BLOCK _UA_GetLocalizedTextResult
  VAR_INPUT
    Enable : BOOL;
  END_VAR
  VAR_OUTPUT
    Done : BOOL;
  END_VAR
  VAR_INPUT
    LocalizedText : UALocalizedText;
  END_VAR
  VAR_OUTPUT
    Locale : _UALocaleType;
    Text : STRING;
  END_VAR

IF Enable=TRUE THEN
	Locale:=LocalizedText.Locale;
	Text:=LocalizedText.Text;
	Done:=TRUE;
END_IF;
IF Enable=FALSE THEN
	Done:=FALSE;
END_IF;
          
END_FUNCTION_BLOCK

FUNCTION_BLOCK _UA_GetArrayDimesionResult
  VAR_INPUT
    Enable : BOOL;
  END_VAR
  VAR_OUTPUT
    Done : BOOL;
  END_VAR
  VAR_INPUT
    ArrayDimension : _UA_UDINT_ArrayType;
    Index : UINT;
  END_VAR
  VAR_OUTPUT
    ArrayDimensionResult : UDINT;
  END_VAR

IF Enable=TRUE THEN
	ArrayDimensionResult:=ArrayDimension.Elements[Index];
	Done:=TRUE;
END_IF;
IF Enable=FALSE THEN
	Done:=FALSE;
END_IF;
          
END_FUNCTION_BLOCK

FUNCTION_BLOCK _UA_GetNodeIDResult
  VAR_INPUT
    Enable : BOOL;
  END_VAR
  VAR_OUTPUT
    Done : BOOL;
  END_VAR
  VAR_INPUT
    NodeID : UANODEID;
  END_VAR
  VAR_OUTPUT
    NamespaceIndex : UINT;
    IdentifierType : UAIdentifierType;
    Identifier : STRING;
  END_VAR

IF Enable=TRUE THEN
	NamespaceIndex:=NodeID.NamespaceIndex;
	IdentifierType:=NodeID.IdentifierType;
	Identifier:=NodeID.Identifier;
	Done:=TRUE;
END_IF;
IF Enable=FALSE THEN
	Done:=FALSE;
END_IF;
          
END_FUNCTION_BLOCK

FUNCTION_BLOCK _UA_GetLocaleResult
  VAR_INPUT
    Enable : BOOL;
  END_VAR
  VAR_OUTPUT
    Done : BOOL;
  END_VAR
  VAR_INPUT
    Locale : _UALocaleType;
    Index : UINT;
  END_VAR
  VAR_OUTPUT
    LocaleResult : STRING;
  END_VAR

IF Enable=TRUE THEN
	LocaleResult:=Locale.Locale[Index];
	Done:=TRUE;
END_IF;
IF Enable=FALSE THEN
	Done:=FALSE;
END_IF;
          
END_FUNCTION_BLOCK

FUNCTION_BLOCK _UA_GetVariableValue
  VAR_INPUT
    Enable : BOOL;
  END_VAR
  VAR_OUTPUT
    Done : BOOL;
  END_VAR
  VAR
    Trigm1 : BOOL;
    Trigged : BOOL;
  END_VAR
  VAR_INPUT
    Index : UINT;
    Variables : _UA_STRING_ArrayType;
  END_VAR
  VAR_OUTPUT
    Result : STRING;
  END_VAR

IF Enable=TRUE THEN
	Result := Variables.Elements[index];
	Done := TRUE;
END_IF;
IF Enable=FALSE THEN
	Done:=FALSE;
END_IF;
          
END_FUNCTION_BLOCK

FUNCTION_BLOCK _UA_GetVariableArray
  VAR_INPUT
    Enable : BOOL;
  END_VAR
  VAR_OUTPUT
    Done : BOOL;
  END_VAR
  VAR_OUTPUT
    Variables : _UA_STRING_ArrayType;
  END_VAR
  VAR_INPUT
    Variable1 : STRING;
    Variable2 : STRING;
    Variable3 : STRING;
    Variable4 : STRING;
    Variable5 : STRING;
    Variable6 : STRING;
    Variable7 : STRING;
    Variable8 : STRING;
    Variable9 : STRING;
    Variable10 : STRING;
    Variable11 : STRING;
    Variable12 : STRING;
    Variable13 : STRING;
    Variable14 : STRING;
    Variable15 : STRING;
    Variable16 : STRING;
    Variable17 : STRING;
    Variable18 : STRING;
    Variable19 : STRING;
    Variable20 : STRING;
  END_VAR

IF Enable=TRUE THEN
	Variables.Elements[1] := Variable1;
	Variables.Elements[2] := Variable2;
	Variables.Elements[3] := Variable3;
	Variables.Elements[4] := Variable4;
	Variables.Elements[5] := Variable5;
	Variables.Elements[6] := Variable6;
	Variables.Elements[7] := Variable7;
	Variables.Elements[8] := Variable8;
	Variables.Elements[9] := Variable9;
	Variables.Elements[10] := Variable10;
	Variables.Elements[11] := Variable11;
	Variables.Elements[12] := Variable12;
	Variables.Elements[13] := Variable13;
	Variables.Elements[14] := Variable14;
	Variables.Elements[15] := Variable15;
	Variables.Elements[16] := Variable16;
	Variables.Elements[17] := Variable17;
	Variables.Elements[18] := Variable18;
	Variables.Elements[19] := Variable19;
	Variables.Elements[20] := Variable20;
	Done:=TRUE;
END_IF;
IF Enable=FALSE THEN
	Done:=FALSE;
END_IF;
          
END_FUNCTION_BLOCK

FUNCTION_BLOCK _UA_GetMonitoringParameter
  VAR_INPUT
    Enable : BOOL;
  END_VAR
  VAR_OUTPUT
    Done : BOOL;
  END_VAR
  VAR_INPUT
    SamplingInterval : STRING;
    QueueSize : UINT;
    DiscardOldest : BOOL;
    DeadbandType : UADeadbandType;
    Deadband : REAL;
  END_VAR
  VAR_OUTPUT
    MonitoringParameter : UAMONITORINGPARAMETER;
  END_VAR

IF Enable=TRUE THEN
	MonitoringParameter.SamplingInterval:=SamplingInterval;
	MonitoringParameter.QueueSize:=QueueSize;
	MonitoringParameter.DiscardOldest:=DiscardOldest;
	MonitoringParameter.DeadbandType:=DeadbandType;
	MonitoringParameter.Deadband:=Deadband;
	Done:=TRUE;
END_IF;
IF Enable=FALSE THEN
	Done:=FALSE;
END_IF;
          
END_FUNCTION_BLOCK

FUNCTION_BLOCK _UA_GetMonitoringParameterArray
  VAR_INPUT
    Enable : BOOL;
  END_VAR
  VAR_OUTPUT
    Done : BOOL;
  END_VAR
  VAR_OUTPUT
    MonitoringParameters : _UA_MONITORINGPARAMETER_ArrayType;
  END_VAR
  VAR_INPUT
    MonitoringParameter1 : UAMONITORINGPARAMETER;
    MonitoringParameter2 : UAMONITORINGPARAMETER;
    MonitoringParameter3 : UAMONITORINGPARAMETER;
    MonitoringParameter4 : UAMONITORINGPARAMETER;
    MonitoringParameter5 : UAMONITORINGPARAMETER;
    MonitoringParameter6 : UAMONITORINGPARAMETER;
    MonitoringParameter7 : UAMONITORINGPARAMETER;
    MonitoringParameter8 : UAMONITORINGPARAMETER;
    MonitoringParameter9 : UAMONITORINGPARAMETER;
    MonitoringParameter10 : UAMONITORINGPARAMETER;
    MonitoringParameter11 : UAMONITORINGPARAMETER;
    MonitoringParameter12 : UAMONITORINGPARAMETER;
    MonitoringParameter13 : UAMONITORINGPARAMETER;
    MonitoringParameter14 : UAMONITORINGPARAMETER;
    MonitoringParameter15 : UAMONITORINGPARAMETER;
    MonitoringParameter16 : UAMONITORINGPARAMETER;
    MonitoringParameter17 : UAMONITORINGPARAMETER;
    MonitoringParameter18 : UAMONITORINGPARAMETER;
    MonitoringParameter19 : UAMONITORINGPARAMETER;
    MonitoringParameter20 : UAMONITORINGPARAMETER;
  END_VAR

IF Enable=TRUE THEN
	MonitoringParameters.Elements[1]:=MonitoringParameter1;
	MonitoringParameters.Elements[2]:=MonitoringParameter2;
	MonitoringParameters.Elements[3]:=MonitoringParameter3;
	MonitoringParameters.Elements[4]:=MonitoringParameter4;
	MonitoringParameters.Elements[5]:=MonitoringParameter5;
	MonitoringParameters.Elements[6]:=MonitoringParameter6;
	MonitoringParameters.Elements[7]:=MonitoringParameter7;
	MonitoringParameters.Elements[8]:=MonitoringParameter8;
	MonitoringParameters.Elements[9]:=MonitoringParameter9;
	MonitoringParameters.Elements[10]:=MonitoringParameter10;
	MonitoringParameters.Elements[11]:=MonitoringParameter11;
	MonitoringParameters.Elements[12]:=MonitoringParameter12;
	MonitoringParameters.Elements[13]:=MonitoringParameter13;
	MonitoringParameters.Elements[14]:=MonitoringParameter14;
	MonitoringParameters.Elements[15]:=MonitoringParameter15;
	MonitoringParameters.Elements[16]:=MonitoringParameter16;
	MonitoringParameters.Elements[17]:=MonitoringParameter17;
	MonitoringParameters.Elements[18]:=MonitoringParameter18;
	MonitoringParameters.Elements[19]:=MonitoringParameter19;
	MonitoringParameters.Elements[20]:=MonitoringParameter20;
	Done:=TRUE;
END_IF;
IF Enable=FALSE THEN
	Done:=FALSE;
END_IF;
          
END_FUNCTION_BLOCK

FUNCTION_BLOCK _UA_GetMethodArgument
  VAR_INPUT
    Enable : BOOL;
    VariantType : _UA_VariantType;
    Value : STRING;
  END_VAR
  VAR_OUTPUT
    MethodArgument : _UA_METHODARGUMENT;
    Done : BOOL;
  END_VAR

IF Enable=TRUE THEN
	MethodArgument.VariantType := VariantType;
	MethodArgument.Value := Value;
	Done:=TRUE;
END_IF;
IF Enable=FALSE THEN
	Done:=FALSE;
END_IF;
          
END_FUNCTION_BLOCK

FUNCTION_BLOCK _UA_GetValuesFromMethodArgument
  VAR_INPUT
    Enable : BOOL;
  END_VAR
  VAR_OUTPUT
    VariantType : _UA_VariantType;
    Value : STRING;
  END_VAR
  VAR_INPUT
    MethodArgument : _UA_METHODARGUMENT;
  END_VAR
  VAR_OUTPUT
    Done : BOOL;
  END_VAR

IF Enable=TRUE THEN
	VariantType := MethodArgument.VariantType;
	Value := MethodArgument.Value;
	Done:=TRUE;
END_IF;
IF Enable=FALSE THEN
	Done:=FALSE;
END_IF;
          
END_FUNCTION_BLOCK

FUNCTION_BLOCK _UA_GetMethodParameter
  VAR_INPUT
    Enable : BOOL;
  END_VAR
  VAR_OUTPUT
    Done : BOOL;
  END_VAR
  VAR_INPUT
    NoOfArgument : UINT;
    Arguments : _UA_METHODARGUMENT_ArrayType;
  END_VAR
  VAR_OUTPUT
    MethodParameter : _UA_MethodParameter;
  END_VAR

IF Enable=TRUE THEN
	MethodParameter.NoOfArgument := NoOfArgument;
	MethodParameter.Arguments := Arguments;
	Done:=TRUE;
END_IF;
IF Enable=FALSE THEN
	Done:=FALSE;
END_IF;
          
END_FUNCTION_BLOCK

FUNCTION_BLOCK _UA_GetValuesFromMethodParameter
  VAR_INPUT
    Enable : BOOL;
  END_VAR
  VAR_OUTPUT
    Done : BOOL;
  END_VAR
  VAR_OUTPUT
    NoOfArgument : UINT;
    Arguments : _UA_METHODARGUMENT_ArrayType;
  END_VAR
  VAR_INPUT
    MethodParameter : _UA_MethodParameter;
  END_VAR

IF Enable=TRUE THEN
	NoOfArgument := MethodParameter.NoOfArgument;
	Arguments := MethodParameter.Arguments;
	Done:=TRUE;
END_IF;
IF Enable=FALSE THEN
	Done:=FALSE;
END_IF;
          
END_FUNCTION_BLOCK

FUNCTION_BLOCK _UA_GetMethodArgumentArray
  VAR_INPUT
    Enable : BOOL;
  END_VAR
  VAR_OUTPUT
    Done : BOOL;
  END_VAR
  VAR_OUTPUT
    MethodArgumentArray : _UA_METHODARGUMENT_ArrayType;
  END_VAR
  VAR_INPUT
    MethodArgument1 : _UA_METHODARGUMENT;
    MethodArgument2 : _UA_METHODARGUMENT;
    MethodArgument3 : _UA_METHODARGUMENT;
    MethodArgument4 : _UA_METHODARGUMENT;
    MethodArgument5 : _UA_METHODARGUMENT;
    MethodArgument6 : _UA_METHODARGUMENT;
    MethodArgument7 : _UA_METHODARGUMENT;
    MethodArgument8 : _UA_METHODARGUMENT;
    MethodArgument9 : _UA_METHODARGUMENT;
    MethodArgument10 : _UA_METHODARGUMENT;
    MethodArgument11 : _UA_METHODARGUMENT;
    MethodArgument12 : _UA_METHODARGUMENT;
    MethodArgument13 : _UA_METHODARGUMENT;
    MethodArgument14 : _UA_METHODARGUMENT;
    MethodArgument15 : _UA_METHODARGUMENT;
    MethodArgument16 : _UA_METHODARGUMENT;
    MethodArgument17 : _UA_METHODARGUMENT;
    MethodArgument18 : _UA_METHODARGUMENT;
    MethodArgument19 : _UA_METHODARGUMENT;
    MethodArgument20 : _UA_METHODARGUMENT;
  END_VAR

IF Enable=TRUE THEN
	MethodArgumentArray.Elements[1] := MethodArgument1;
	MethodArgumentArray.Elements[2] := MethodArgument2;
	MethodArgumentArray.Elements[3] := MethodArgument3;
	MethodArgumentArray.Elements[4] := MethodArgument4;
	MethodArgumentArray.Elements[5] := MethodArgument5;
	MethodArgumentArray.Elements[6] := MethodArgument6;
	MethodArgumentArray.Elements[7] := MethodArgument7;
	MethodArgumentArray.Elements[8] := MethodArgument8;
	MethodArgumentArray.Elements[9] := MethodArgument9;
	MethodArgumentArray.Elements[10] := MethodArgument10;
	MethodArgumentArray.Elements[11] := MethodArgument11;
	MethodArgumentArray.Elements[12] := MethodArgument12;
	MethodArgumentArray.Elements[13] := MethodArgument13;
	MethodArgumentArray.Elements[14] := MethodArgument14;
	MethodArgumentArray.Elements[15] := MethodArgument15;
	MethodArgumentArray.Elements[16] := MethodArgument16;
	MethodArgumentArray.Elements[17] := MethodArgument17;
	MethodArgumentArray.Elements[18] := MethodArgument18;
	MethodArgumentArray.Elements[19] := MethodArgument19;
	MethodArgumentArray.Elements[20] := MethodArgument20;
	Done:=TRUE;
END_IF;
IF Enable=FALSE THEN
	Done:=FALSE;
END_IF;
          
END_FUNCTION_BLOCK

FUNCTION_BLOCK _UA_GetMethodArgumentFromArray
  VAR_INPUT
    Enable : BOOL;
  END_VAR
  VAR_OUTPUT
    Done : BOOL;
  END_VAR
  VAR_INPUT
    Index : UINT;
    MethodArgumentArray : _UA_METHODARGUMENT_ArrayType;
  END_VAR
  VAR_OUTPUT
    MethodArgument : _UA_METHODARGUMENT;
  END_VAR

IF Enable=TRUE THEN
	MethodArgument := MethodArgumentArray.Elements[Index];
	Done:=TRUE;
END_IF;
IF Enable=FALSE THEN
	Done:=FALSE;
END_IF;
          
END_FUNCTION_BLOCK

FUNCTION_BLOCK _UA_GetMonitoredItemVariableValue
  VAR_INPUT
    Enable : BOOL;
  END_VAR
  VAR_OUTPUT
    Done : BOOL;
    Busy : BOOL;
  END_VAR
  VAR_INPUT
    GlobalIndex : UINT;
    LocalIndex : UINT;
  END_VAR
  VAR_OUTPUT
    Value : STRING;
  END_VAR
  VAR
    Trigged : BOOL;
    State : DWORD;
  END_VAR

{{
  #ifdef _ENABLE_OPC_UA_CLIENT
  extern void ___UA_GetMonitoredItemVariableValueFB(_UA_GETMONITOREDITEMVARIABLEVALUE*);
  ___UA_GetMonitoredItemVariableValueFB(data__);
  #endif
}}
          
END_FUNCTION_BLOCK

FUNCTION_BLOCK _UA_GetMonitoredItemValuesChangedValue
  VAR_INPUT
    Enable : BOOL;
  END_VAR
  VAR_OUTPUT
    Done : BOOL;
    Busy : BOOL;
  END_VAR
  VAR_INPUT
    GlobalIndex : UINT;
    LocalIndex : UINT;
  END_VAR
  VAR_OUTPUT
    ValueChanged : BOOL;
  END_VAR

{{
  #ifdef _ENABLE_OPC_UA_CLIENT
  extern void ___UA_GetMonitoredItemValuesChangedValueFB(_UA_GETMONITOREDITEMVALUESCHANGEDVALUE*);
  ___UA_GetMonitoredItemValuesChangedValueFB(data__);
  #endif
}}
          
END_FUNCTION_BLOCK
